TYPE ST_RejectReason_PK1_OUT3 :
STRUCT
	Reason	:STRING;
END_STRUCT
END_TYPE

(* stored: Version 1.1.0.1, ProductVersion 3.1.4024.13
   DUT ST_RejectReason_PK1_OUT3: Id {1abd13f9-779d-4574-b226-50c84ae7e43d} *)
